INTERFACE I_Stack

METHOD Peek : T_DATA_TYPE
END_METHOD

METHOD Pop
END_METHOD

METHOD Push
VAR_INPUT
		Data 	: T_DATA_TYPE;
END_VAR
END_METHOD

METHOD Show
VAR_INPUT
END_VAR
END_METHOD

END_INTERFACE

(* stored: Version 1.1.0.1, ProductVersion 3.1.4024.4
   Itf I_Stack: Id {9e2aef48-43c6-47a2-99ac-ee56af742825}
   Method Peek: Id {5f4823b8-9f25-4636-ade1-85e0b21e7a3a}
   Method Pop: Id {33f1041c-447f-4e90-a35e-c0d47a2ca3eb}
   Method Push: Id {8a193e74-d1b6-4a14-8325-1c01989906a1}
   Method Show: Id {bb0198e6-609d-4a79-b92f-0f482b881cf5} *)
